FUNCTION_BLOCK FB_FileRingBufferToDB
VAR_INPUT
	udiNovRam_BufferIndex:UDINT;
	udiFile_Index:UDINT;
	dataType:DINT;
END_VAR

IF dataType = E_StructureType.AlarmHistory THEN
	M_AlarmHistory(udiNovRam_BufferIndex:=udiNovRam_BufferIndex,udiFile_Index:=udiFile_Index);
ELSIF dataType = E_StructureType.ProductionHistory THEN
	M_ProductionHistory(udiNovRam_BufferIndex:=udiNovRam_BufferIndex,udiFile_Index:=udiFile_Index);
ELSIF dataType = E_StructureType.ProductionReport THEN
	M_ProductionReport(udiNovRam_BufferIndex:=udiNovRam_BufferIndex,udiFile_Index:=udiFile_Index);
ELSIF dataType = E_StructureType.ProductionSummary THEN
	M_ProductionSummary(udiNovRam_BufferIndex:=udiNovRam_BufferIndex,udiFile_Index:=udiFile_Index);
ELSIF dataType = E_StructureType.SoDuration THEN
	M_SoDuration(udiNovRam_BufferIndex:=udiNovRam_BufferIndex,udiFile_Index:=udiFile_Index);
ELSIF dataType = E_StructureType.StopCount THEN
	M_StopCount(udiNovRam_BufferIndex:=udiNovRam_BufferIndex,udiFile_Index:=udiFile_Index);
ELSIF dataType = E_StructureType.RegularCheckResults THEN
	M_RegularCheckResults(udiNovRam_BufferIndex:=udiNovRam_BufferIndex,udiFile_Index:=udiFile_Index);
END_IF

METHOD M_AlarmHistory : BOOL
VAR_INPUT
	
	//udiFileNo:UDINT;
	udiNovRam_BufferIndex:UDINT;
	udiFile_Index:UDINT;
END_VAR
VAR_INST
	arrDataFromFile:ARRAY[0..GVL.arrArrayLength[E_StructureType.AlarmHistory]-1] OF ST_AlarmInfo_DB_save;
	DataToDB:ST_AlarmInfo_DB_save;
	AnalizeIndex:UDINT;//should be kept by NovRam
	iStep:INT;
	i:UDINT;
	fbFileRingBuffer: FB_FileRingBuffer := ( sNetId     := '',
                                             sPathName  := '',
                                             ePath      := PATH_GENERIC,
                                             nID        := 1,
                                             cbBuffer   := gvl.arrFileRingBufferSize[E_StructureType.AlarmHistory], //5MB(5*10^6Bytes)
                                             bOverwrite := FALSE,
                                             pWriteBuff := 0,
                                             cbWriteLen := 0,
                                             pReadBuff  := 0,
                                             cbReadLen  := 0,
                                             tTimeout   := T#1S );
	bBusy:BOOL;
	bError:BOOL;
	nErrID:UDINT;
	stHeader:ST_FileRBufferHead;
    //loadData  : ARRAY[0..511] OF BYTE :=[512(0)];
    //cbLoad    : UDINT;
	
	fileName: STRING(255);
	eStrIndex:DINT;
	fbAlarmHistory_DB		: FB_AlarmHistory_DB;
END_VAR
//Config
eStrIndex:=E_StructureType.AlarmHistory;

fbFileRingBuffer(sPathName:=fileName
				,bBusy=>bBusy,bError=>bError,nErrID=>nErrID
				,stHeader=>stHeader);
//DB_Test
fbAlarmHistory_DB(udiDBID:=1);

CASE iStep OF
	0://check if file full 
		IF gvl.NovRamData.arrFileRingBuffer_Status[eStrIndex].bFileFull[udiNovRam_BufferIndex][udiFile_Index] = TRUE//file full = should work 
		THEN
			
			fileName:=M_GetFileName(structureType:=eStrIndex
									,udiNovRam_BufferIndex:=udiNovRam_BufferIndex
									,udiFile_Index:=udiFile_Index);
			
			iStep:=100;
		END_IF
	100:// Open file
		
		AnalizeIndex:=0;
		fbFileRingBuffer.A_Open();
		
		iStep:=200;
	200://wait done / read head
		IF NOT fbFileRingBuffer.bBusy AND NOT fbFileRingBuffer.bError THEN
			
			fbFileRingBuffer.A_GetHead(pReadBuff := ADR(arrDataFromFile), cbReadLen := SIZEOF(arrDataFromFile));
			
			iStep:=300;
		END_IF
	300://wait done / take data from array
		IF NOT fbFileRingBuffer.bBusy AND NOT fbFileRingBuffer.bError THEN
			
			DataToDB:=arrDataFromFile[AnalizeIndex];
			
			iStep:=310;
		ELSIF NOT fbFileRingBuffer.bBusy AND fbFileRingBuffer.bError THEN//Empty
			iStep:=600;
		END_IF
	310:// write to DB
	
		//write DataToDB to DB
		DataToDB.lrTime_ms    	:= 987;
		DataToDB.diMsgNumber  	:= 777;
		DataToDB.sTimeString 	:= '2023-11-24 17:17:17';
		DataToDB.wsMsgText    	:= "TEST_MsgText軟體測試";
		DataToDB.sPLC        	:= 'CoreSysTest';
		DataToDB.wsEquipment  	:= "RSA軟體測試";
		DataToDB.sFaam_id    	:= 'TEST_Faam_id';
		
		IF fbAlarmHistory_DB.M_Upload(stAlarmInfo:=DataToDB) THEN
			iStep:=320;
		END_IF
		
	320://wait done
		
		IF NOT fbAlarmHistory_DB.bError THEN//write OK
		
			AnalizeIndex:=AnalizeIndex+1;
			
			iStep:=330;
			
		ELSE//write failed need to write to log
			;
		END_IF
		
	330://Check if all data in array Analized
		IF AnalizeIndex < GVL.arrArrayLength[eStrIndex] THEN//not done
			iStep:=300;//go back
		ELSE//array data done
			iStep:=400;//complete this array
		END_IF
		
	400://wait done / remove Head
	
		fbFileRingBuffer.A_RemoveHead(pReadBuff := ADR(arrDataFromFile), cbReadLen := SIZEOF(arrDataFromFile));
		
		iStep:=500;
		
	500://wait done / check if all data got?
		IF NOT fbFileRingBuffer.bBusy AND NOT fbFileRingBuffer.bError THEN
			IF stHeader.nCount > 0 THEN
				iStep:=100;//Go Back
			ELSE
				iStep:=600;//finish
			END_IF
		END_IF
	600://reset file
	
		fbFileRingBuffer.A_Reset();
		
		iStep:=700;
		
	700://wait done / close file
		IF NOT fbFileRingBuffer.bBusy AND NOT fbFileRingBuffer.bError THEN
			
			fbFileRingBuffer.A_Close();
			
			iStep:=800;
		END_IF
	800://wait done
		IF NOT fbFileRingBuffer.bBusy AND NOT fbFileRingBuffer.bError THEN
			
			GVL.NovRamData.arrFileRingBuffer_Status[eStrIndex].bFileFull[udiNovRam_BufferIndex][udiFile_Index]:=FALSE;
			
			iStep:=0;
			
		END_IF
		
	
END_CASE
END_METHOD

METHOD M_GetFileName : STRING(255)
VAR_INPUT
	structureType:DINT;
	udiNovRam_BufferIndex:UDINT;
	udiFile_Index:UDINT;
END_VAR
VAR
	tempString:STRING(255);
	tempString2:STRING(255);
	tempFileNo:UDINT;
END_VAR
IF structureType=E_StructureType.AlarmHistory THEN
	tempString:=CONCAT(gvl.arrfileFolder[structureType],'AlarmHistory');
ELSIF structureType=E_StructureType.ProductionHistory THEN
	tempString:=CONCAT(gvl.arrfileFolder[structureType],'ProductionHistory');
ELSIF structureType=E_StructureType.ProductionReport THEN
	tempString:=CONCAT(gvl.arrfileFolder[structureType],'ProductionReport');
	ELSIF structureType=E_StructureType.ProductionSummary THEN
	tempString:=CONCAT(gvl.arrfileFolder[structureType],'ProductionSummary');
ELSIF structureType=E_StructureType.SoDuration THEN
	tempString:=CONCAT(gvl.arrfileFolder[structureType],'SoDuration');
ELSIF structureType=E_StructureType.StopCount THEN
	tempString:=CONCAT(gvl.arrfileFolder[structureType],'StopCount');
ELSIF structureType=E_StructureType.RegularCheckResults THEN
	tempString:=CONCAT(gvl.arrfileFolder[structureType],'RegularCheckResults');
END_IF

tempFileNo:=(udiNovRam_BufferIndex) * GVL.FileRingBufferRatio + (udiFile_Index + 1);
tempString2:=CONCAT(tempString,UDINT_TO_STRING(tempFileNo));
M_GetFileName:=CONCAT(tempString2,'.dat');
END_METHOD

{warning 'add method implementation '}
METHOD M_ProductionHistory : BOOL
VAR_INPUT
	
	//udiFileNo:UDINT;
	udiNovRam_BufferIndex:UDINT;
	udiFile_Index:UDINT;
END_VAR
VAR_INST
	arrDataFromFile:ARRAY[0..GVL.arrArrayLength[E_StructureType.ProductionHistory]-1] OF ST_Production_History_DB_Test;
	DataToDB:ST_Production_History_DB_Test;
	AnalizeIndex:UDINT;//should be kept by NovRam
	iStep:INT;
	i:UDINT;
	fbFileRingBuffer: FB_FileRingBuffer := ( sNetId     := '',
                                             sPathName  := '',
                                             ePath      := PATH_GENERIC,
                                             nID        := 1,
                                             cbBuffer   := gvl.arrFileRingBufferSize[E_StructureType.ProductionHistory], //5MB(5*10^6Bytes)
                                             bOverwrite := FALSE,
                                             pWriteBuff := 0,
                                             cbWriteLen := 0,
                                             pReadBuff  := 0,
                                             cbReadLen  := 0,
                                             tTimeout   := T#1S );
	bBusy:BOOL;
	bError:BOOL;
	nErrID:UDINT;
	stHeader:ST_FileRBufferHead;
    //loadData  : ARRAY[0..511] OF BYTE :=[512(0)];
    //cbLoad    : UDINT;
	
	fileName: STRING(255);
	eStrIndex:DINT;
	
	//DB
	fbProductionHistoryInspection_DB		: FB_ProductionHistoryInspection_DB;
	PHI_GroupData_DB : ST_PHI_GroupData_DB;
END_VAR
//Config
eStrIndex:=E_StructureType.ProductionHistory;

fbFileRingBuffer(sPathName:=fileName
				,bBusy=>bBusy,bError=>bError,nErrID=>nErrID
				,stHeader=>stHeader);
				
//DB_Test
fbProductionHistoryInspection_DB(udiDBID:=1);

CASE iStep OF
	0://check if file full 
		IF gvl.NovRamData.arrFileRingBuffer_Status[eStrIndex].bFileFull[udiNovRam_BufferIndex][udiFile_Index] = TRUE//file full = should work 
		THEN
			
			fileName:=M_GetFileName(structureType:=eStrIndex
									,udiNovRam_BufferIndex:=udiNovRam_BufferIndex
									,udiFile_Index:=udiFile_Index);
			
			iStep:=100;
		END_IF
	100:// Open file
		
		AnalizeIndex:=0;
		fbFileRingBuffer.A_Open();
		
		iStep:=200;
	200://wait done / read head
		IF NOT fbFileRingBuffer.bBusy AND NOT fbFileRingBuffer.bError THEN
			
			fbFileRingBuffer.A_GetHead(pReadBuff := ADR(arrDataFromFile), cbReadLen := SIZEOF(arrDataFromFile));
			
			iStep:=300;
		END_IF
	300://wait done / take data from array
		IF NOT fbFileRingBuffer.bBusy AND NOT fbFileRingBuffer.bError THEN
			
			DataToDB:=arrDataFromFile[AnalizeIndex];
			
			iStep:=310;
		ELSIF NOT fbFileRingBuffer.bBusy AND fbFileRingBuffer.bError THEN//Empty
			iStep:=600;
		END_IF
	310:// write to DB
	
		//write DataToDB to DB
		DataToDB.rDuration    	:= 987;
		DataToDB.usiStation_number  	:= 87;
		DataToDB.sStation_name 	:= 'Station Test';
		DataToDB.sFaam_id    	:= 'TEST_Faam_id';
		
		PHI_GroupData_DB.stProductHistory.dtStart_time 			:= TIME_TO_DT(TIME());
		PHI_GroupData_DB.stProductHistory.dtEnd_time 				:= TIME_TO_DT(TIME());
		PHI_GroupData_DB.stProductHistory.rDuration 				:= TIME_TO_REAL(TIME()) / 1000; // ms to s
		PHI_GroupData_DB.stProductHistory.diStation_number 		:= 1;	// index id
		PHI_GroupData_DB.stProductHistory.wsStation_name 			:= "TEST_Station1";		// index name from DB.HC
		PHI_GroupData_DB.stProductHistory.diTrack_number 			:= 1;	//20230106 改為hardcode 1
		PHI_GroupData_DB.stProductHistory.bPart_ok_overal_results := TRUE;
		PHI_GroupData_DB.stProductHistory.sSo_number 				:= 'Fred';				// From ADS  //需要對應DB的So表的So_Number
		PHI_GroupData_DB.stProductHistory.sFaam_id 				:= 'FB000120-E002-0001';		// from DB
		PHI_GroupData_DB.stProductHistory.diSo_id 				:= 3736;			// from ADS  //需要對應DB的So表So_id
		PHI_GroupData_DB.stProductHistory.diWpc_number			:= 2; // ShuttleID
		
		IF fbProductionHistoryInspection_DB.M_Upload(stPHI:=PHI_GroupData_DB) THEN
			iStep:=320;
		END_IF
		
	320://wait done
		
		IF NOT fbProductionHistoryInspection_DB.bError THEN//write OK
		
			AnalizeIndex:=AnalizeIndex+1;
			
			iStep:=330;
			
		ELSE//write failed need to write to log
			;
		END_IF
		
	330://Check if all data in array Analized
		IF AnalizeIndex < GVL.arrArrayLength[eStrIndex] THEN//not done
			iStep:=300;//go back
		ELSE//array data done
			iStep:=400;//complete this array
		END_IF
		
	400://wait done / remove Head
	
		fbFileRingBuffer.A_RemoveHead(pReadBuff := ADR(arrDataFromFile), cbReadLen := SIZEOF(arrDataFromFile));
		
		iStep:=500;
		
	500://wait done / check if all data got?
		IF NOT fbFileRingBuffer.bBusy AND NOT fbFileRingBuffer.bError THEN
			IF stHeader.nCount > 0 THEN
				iStep:=100;//Go Back
			ELSE
				iStep:=600;//finish
			END_IF
		END_IF
	600://reset file
	
		fbFileRingBuffer.A_Reset();
		
		iStep:=700;
		
	700://wait done / close file
		IF NOT fbFileRingBuffer.bBusy AND NOT fbFileRingBuffer.bError THEN
			
			fbFileRingBuffer.A_Close();
			
			iStep:=800;
		END_IF
	800://wait done
		IF NOT fbFileRingBuffer.bBusy AND NOT fbFileRingBuffer.bError THEN
			
			GVL.NovRamData.arrFileRingBuffer_Status[eStrIndex].bFileFull[udiNovRam_BufferIndex][udiFile_Index]:=FALSE;
			
			iStep:=0;
			
		END_IF
		
	
END_CASE
END_METHOD

METHOD M_ProductionReport : BOOL
VAR_INPUT
	
	//udiFileNo:UDINT;
	udiNovRam_BufferIndex:UDINT;
	udiFile_Index:UDINT;
END_VAR
VAR_INST
	arrDataFromFile:ARRAY[0..GVL.arrArrayLength[E_StructureType.ProductionReport]-1] OF ST_OEE_ProductionReport;
	DataToDB:ST_OEE_ProductionReport;
	AnalizeIndex:UDINT;//should be kept by NovRam
	iStep:INT;
	i:UDINT;
	fbFileRingBuffer: FB_FileRingBuffer := ( sNetId     := '',
                                             sPathName  := '',
                                             ePath      := PATH_GENERIC,
                                             nID        := 1,
                                             cbBuffer   := gvl.arrFileRingBufferSize[E_StructureType.ProductionReport], //5MB(5*10^6Bytes)
                                             bOverwrite := FALSE,
                                             pWriteBuff := 0,
                                             cbWriteLen := 0,
                                             pReadBuff  := 0,
                                             cbReadLen  := 0,
                                             tTimeout   := T#1S );
	bBusy:BOOL;
	bError:BOOL;
	nErrID:UDINT;
	stHeader:ST_FileRBufferHead;
    //loadData  : ARRAY[0..511] OF BYTE :=[512(0)];
    //cbLoad    : UDINT;
	
	fileName: STRING(255);
	eStrIndex:DINT;
	fbOEE_ProductionReport_DB:FB_OEE_ProductionReport_DB;
END_VAR
//Config
eStrIndex:=E_StructureType.ProductionReport;

fbFileRingBuffer(sPathName:=fileName
				,bBusy=>bBusy,bError=>bError,nErrID=>nErrID
				,stHeader=>stHeader);
				
CASE iStep OF
	0://check if file full 
		IF gvl.NovRamData.arrFileRingBuffer_Status[eStrIndex].bFileFull[udiNovRam_BufferIndex][udiFile_Index] = TRUE//file full = should work 
		THEN
			
			fileName:=M_GetFileName(structureType:=eStrIndex
									,udiNovRam_BufferIndex:=udiNovRam_BufferIndex
									,udiFile_Index:=udiFile_Index);
			
			iStep:=100;
		END_IF
	100:// Open file
		
		AnalizeIndex:=0;
		fbFileRingBuffer.A_Open();
		
		iStep:=200;
	200://wait done / read head
		IF NOT fbFileRingBuffer.bBusy AND NOT fbFileRingBuffer.bError THEN
			
			fbFileRingBuffer.A_GetHead(pReadBuff := ADR(arrDataFromFile), cbReadLen := SIZEOF(arrDataFromFile));
			
			iStep:=300;
		END_IF
	300://wait done / take data from array
		IF NOT fbFileRingBuffer.bBusy AND NOT fbFileRingBuffer.bError THEN
			
			DataToDB:=arrDataFromFile[AnalizeIndex];
			
			iStep:=310;
		ELSIF NOT fbFileRingBuffer.bBusy AND fbFileRingBuffer.bError THEN//Empty
			iStep:=600;
		END_IF
	310:// write to DB
	
		//write DataToDB to DB
		DataToDB.diOk_part_count:=123;
		DataToDB.sSo_number                    	:= 'Fred';
		DataToDB.sFaam_id                      	:= 'FB000120-E002-0001';
		DataToDB.diSo_id                        := 3736;
		
		IF fbOEE_ProductionReport_DB.M_Upload(stOeeProductionReport:=DataToDB) THEN
			iStep:=320;
		END_IF
		
	320://wait done
		
			IF NOT fbOEE_ProductionReport_DB.bError THEN//write OK
			
				AnalizeIndex:=AnalizeIndex+1;
				
				iStep:=330;
				
			ELSE//write failed need to write to log
				;
			END_IF
		
		
	330://Check if all data in array Analized
		IF AnalizeIndex < GVL.arrArrayLength[eStrIndex] THEN//not done
			iStep:=300;//go back
		ELSE//array data done
			iStep:=400;//complete this array
		END_IF
		
	400://wait done / remove Head
	
		fbFileRingBuffer.A_RemoveHead(pReadBuff := ADR(arrDataFromFile), cbReadLen := SIZEOF(arrDataFromFile));
		
		iStep:=500;
		
	500://wait done / check if all data got?
		IF NOT fbFileRingBuffer.bBusy AND NOT fbFileRingBuffer.bError THEN
			IF stHeader.nCount > 0 THEN
				iStep:=100;//Go Back
			ELSE
				iStep:=600;//finish
			END_IF
		END_IF
	600://reset file
	
		fbFileRingBuffer.A_Reset();
		
		iStep:=700;
		
	700://wait done / close file
		IF NOT fbFileRingBuffer.bBusy AND NOT fbFileRingBuffer.bError THEN
			
			fbFileRingBuffer.A_Close();
			
			iStep:=800;
		END_IF
	800://wait done
		IF NOT fbFileRingBuffer.bBusy AND NOT fbFileRingBuffer.bError THEN
			
			GVL.NovRamData.arrFileRingBuffer_Status[eStrIndex].bFileFull[udiNovRam_BufferIndex][udiFile_Index]:=FALSE;
			
			iStep:=0;
			
		END_IF
		
	
END_CASE
END_METHOD

METHOD M_ProductionSummary : BOOL
VAR_INPUT
	
	//udiFileNo:UDINT;
	udiNovRam_BufferIndex:UDINT;
	udiFile_Index:UDINT;
END_VAR
VAR_INST
	arrDataFromFile:ARRAY[0..GVL.arrArrayLength[E_StructureType.ProductionSummary]-1] OF ST_OEE_ProductionSummary;
	DataToDB:ST_OEE_ProductionSummary;
	AnalizeIndex:UDINT;//should be kept by NovRam
	iStep:INT;
	i:UDINT;
	fbFileRingBuffer: FB_FileRingBuffer := ( sNetId     := '',
                                             sPathName  := '',
                                             ePath      := PATH_GENERIC,
                                             nID        := 1,
                                             cbBuffer   := gvl.arrFileRingBufferSize[E_StructureType.ProductionSummary], //5MB(5*10^6Bytes)
                                             bOverwrite := FALSE,
                                             pWriteBuff := 0,
                                             cbWriteLen := 0,
                                             pReadBuff  := 0,
                                             cbReadLen  := 0,
                                             tTimeout   := T#1S );
	bBusy:BOOL;
	bError:BOOL;
	nErrID:UDINT;
	stHeader:ST_FileRBufferHead;
    //loadData  : ARRAY[0..511] OF BYTE :=[512(0)];
    //cbLoad    : UDINT;
	
	fileName: STRING(255);
	eStrIndex:DINT;
	fbOEE_ProductionSummary_DB:FB_OEE_ProductionSummary_DB;
END_VAR
//Config
eStrIndex:=E_StructureType.ProductionSummary;

fbFileRingBuffer(sPathName:=fileName
				,bBusy=>bBusy,bError=>bError,nErrID=>nErrID
				,stHeader=>stHeader);
				
CASE iStep OF
	0://check if file full 
		IF gvl.NovRamData.arrFileRingBuffer_Status[eStrIndex].bFileFull[udiNovRam_BufferIndex][udiFile_Index] = TRUE//file full = should work 
		THEN
			
			fileName:=M_GetFileName(structureType:=eStrIndex
									,udiNovRam_BufferIndex:=udiNovRam_BufferIndex
									,udiFile_Index:=udiFile_Index);
			
			iStep:=100;
		END_IF
	100:// Open file
		
		AnalizeIndex:=0;
		fbFileRingBuffer.A_Open();
		
		iStep:=200;
	200://wait done / read head
		IF NOT fbFileRingBuffer.bBusy AND NOT fbFileRingBuffer.bError THEN
			
			fbFileRingBuffer.A_GetHead(pReadBuff := ADR(arrDataFromFile), cbReadLen := SIZEOF(arrDataFromFile));
			
			iStep:=300;
		END_IF
	300://wait done / take data from array
		IF NOT fbFileRingBuffer.bBusy AND NOT fbFileRingBuffer.bError THEN
			
			DataToDB:=arrDataFromFile[AnalizeIndex];
			
			iStep:=310;
		ELSIF NOT fbFileRingBuffer.bBusy AND fbFileRingBuffer.bError THEN//Empty
			iStep:=600;
		END_IF
	310:// write to DB
	
		//write DataToDB to DB
		DataToDB.diSo_id:=123;
		DataToDB.diSummary_value:=456;
		DataToDB.sSo_number                    	:= 'Fred';
		DataToDB.sFaam_id                      	:= 'FB000120-E002-0001';
		DataToDB.diSo_id                        := 3736;
		
		IF fbOEE_ProductionSummary_DB.M_Upload(stOEEProductionSummary:=DataToDB) THEN
			iStep:=320;
		END_IF
		
		
	320://wait done
		
			IF NOT fbOEE_ProductionSummary_DB.bError THEN//write OK
			
				AnalizeIndex:=AnalizeIndex+1;
				
				iStep:=330;
				
			ELSE//write failed need to write to log
				;
			END_IF
		
		
	330://Check if all data in array Analized
		IF AnalizeIndex < GVL.arrArrayLength[eStrIndex] THEN//not done
			iStep:=300;//go back
		ELSE//array data done
			iStep:=400;//complete this array
		END_IF
		
	400://wait done / remove Head
	
		fbFileRingBuffer.A_RemoveHead(pReadBuff := ADR(arrDataFromFile), cbReadLen := SIZEOF(arrDataFromFile));
		
		iStep:=500;
		
	500://wait done / check if all data got?
		IF NOT fbFileRingBuffer.bBusy AND NOT fbFileRingBuffer.bError THEN
			IF stHeader.nCount > 0 THEN
				iStep:=100;//Go Back
			ELSE
				iStep:=600;//finish
			END_IF
		END_IF
	600://reset file
	
		fbFileRingBuffer.A_Reset();
		
		iStep:=700;
		
	700://wait done / close file
		IF NOT fbFileRingBuffer.bBusy AND NOT fbFileRingBuffer.bError THEN
			
			fbFileRingBuffer.A_Close();
			
			iStep:=800;
		END_IF
	800://wait done
		IF NOT fbFileRingBuffer.bBusy AND NOT fbFileRingBuffer.bError THEN
			
			GVL.NovRamData.arrFileRingBuffer_Status[eStrIndex].bFileFull[udiNovRam_BufferIndex][udiFile_Index]:=FALSE;
			
			iStep:=0;
			
		END_IF
		
	
END_CASE
END_METHOD

METHOD M_RegularCheckResults : BOOL
VAR_INPUT
	
	//udiFileNo:UDINT;
	udiNovRam_BufferIndex:UDINT;
	udiFile_Index:UDINT;
END_VAR
VAR_INST
	arrDataFromFile:ARRAY[0..GVL.arrArrayLength[E_StructureType.RegularCheckResults]-1] OF ST_RegularCheck_Results_DB;
	DataToDB:ST_RegularCheck_Results;//TEST
	AnalizeIndex:UDINT;//should be kept by NovRam
	iStep:INT;
	i:UDINT;
	fbFileRingBuffer: FB_FileRingBuffer := ( sNetId     := '',
                                             sPathName  := '',
                                             ePath      := PATH_GENERIC,
                                             nID        := 1,
                                             cbBuffer   := gvl.arrFileRingBufferSize[E_StructureType.RegularCheckResults], //5MB(5*10^6Bytes)
                                             bOverwrite := FALSE,
                                             pWriteBuff := 0,
                                             cbWriteLen := 0,
                                             pReadBuff  := 0,
                                             cbReadLen  := 0,
                                             tTimeout   := T#1S );
	bBusy:BOOL;
	bError:BOOL;
	nErrID:UDINT;
	stHeader:ST_FileRBufferHead;
    //loadData  : ARRAY[0..511] OF BYTE :=[512(0)];
    //cbLoad    : UDINT;
	
	fileName: STRING(255);
	eStrIndex:DINT;
	fbRegular_Check_Results_DB:FB_Regular_Check_Results_DB;
END_VAR
//Config
eStrIndex:=E_StructureType.RegularCheckResults;

fbFileRingBuffer(sPathName:=fileName
				,bBusy=>bBusy,bError=>bError,nErrID=>nErrID
				,stHeader=>stHeader);
				
CASE iStep OF
	0://check if file full 
		IF gvl.NovRamData.arrFileRingBuffer_Status[eStrIndex].bFileFull[udiNovRam_BufferIndex][udiFile_Index] = TRUE//file full = should work 
		THEN
			
			fileName:=M_GetFileName(structureType:=eStrIndex
									,udiNovRam_BufferIndex:=udiNovRam_BufferIndex
									,udiFile_Index:=udiFile_Index);
			
			iStep:=100;
		END_IF
	100:// Open file
		
		AnalizeIndex:=0;
		fbFileRingBuffer.A_Open();
		
		iStep:=200;
	200://wait done / read head
		IF NOT fbFileRingBuffer.bBusy AND NOT fbFileRingBuffer.bError THEN
			
			fbFileRingBuffer.A_GetHead(pReadBuff := ADR(arrDataFromFile), cbReadLen := SIZEOF(arrDataFromFile));
			
			iStep:=300;
		END_IF
	300://wait done / take data from array
		IF NOT fbFileRingBuffer.bBusy AND NOT fbFileRingBuffer.bError THEN
			
			//DataToDB:=arrDataFromFile[AnalizeIndex];
			M_ST_RegularCheckResults_Convert(input:=arrDataFromFile[AnalizeIndex]
											,output=>DataToDB);
			iStep:=310;
		ELSIF NOT fbFileRingBuffer.bBusy AND fbFileRingBuffer.bError THEN//Empty
			iStep:=600;
		END_IF
	310:// write to DB
		
		//write DataToDB to DB
		DataToDB.eSensor:=E_RegularCheckSensorResult.Fail;
		DataToDB.eSensor2:=E_RegularCheckSensorResult.Fail;
		DataToDB.sSo_number                    	:= 'Fred';
		DataToDB.sFaam_id                      	:= 'FB000120-E002-0001';
		DataToDB.diSo_id                        := 3736;
		
		IF fbRegular_Check_Results_DB.M_Upload(stRcResults:=DataToDB) THEN
			iStep:=320;
		END_IF
		
	320://wait done
		
		IF NOT fbRegular_Check_Results_DB.bError THEN//write OK
		
			AnalizeIndex:=AnalizeIndex+1;
			
			iStep:=330;
			
		ELSE//write failed need to write to log
			;
		END_IF
		
	330://Check if all data in array Analized
		IF AnalizeIndex < GVL.arrArrayLength[eStrIndex] THEN//not done
			iStep:=300;//go back
		ELSE//array data done
			iStep:=400;//complete this array
		END_IF
		
	400://wait done / remove Head
	
		fbFileRingBuffer.A_RemoveHead(pReadBuff := ADR(arrDataFromFile), cbReadLen := SIZEOF(arrDataFromFile));
		
		iStep:=500;
		
	500://wait done / check if all data got?
		IF NOT fbFileRingBuffer.bBusy AND NOT fbFileRingBuffer.bError THEN
			IF stHeader.nCount > 0 THEN
				iStep:=100;//Go Back
			ELSE
				iStep:=600;//finish
			END_IF
		END_IF
	600://reset file
	
		fbFileRingBuffer.A_Reset();
		
		iStep:=700;
		
	700://wait done / close file
		IF NOT fbFileRingBuffer.bBusy AND NOT fbFileRingBuffer.bError THEN
			
			fbFileRingBuffer.A_Close();
			
			iStep:=800;
		END_IF
	800://wait done
		IF NOT fbFileRingBuffer.bBusy AND NOT fbFileRingBuffer.bError THEN
			
			GVL.NovRamData.arrFileRingBuffer_Status[eStrIndex].bFileFull[udiNovRam_BufferIndex][udiFile_Index]:=FALSE;
			
			iStep:=0;
			
		END_IF
		
	
END_CASE
END_METHOD

METHOD M_SoDuration : BOOL
VAR_INPUT
	
	//udiFileNo:UDINT;
	udiNovRam_BufferIndex:UDINT;
	udiFile_Index:UDINT;
END_VAR
VAR_INST
	arrDataFromFile:ARRAY[0..GVL.arrArrayLength[E_StructureType.SoDuration]-1] OF ST_SoDuration;
	DataToDB:ST_SoDuration;
	AnalizeIndex:UDINT;//should be kept by NovRam
	iStep:INT;
	i:UDINT;
	fbFileRingBuffer: FB_FileRingBuffer := ( sNetId     := '',
                                             sPathName  := '',
                                             ePath      := PATH_GENERIC,
                                             nID        := 1,
                                             cbBuffer   := gvl.arrFileRingBufferSize[E_StructureType.ProductionSummary], //5MB(5*10^6Bytes)
                                             bOverwrite := FALSE,
                                             pWriteBuff := 0,
                                             cbWriteLen := 0,
                                             pReadBuff  := 0,
                                             cbReadLen  := 0,
                                             tTimeout   := T#1S );
	bBusy:BOOL;
	bError:BOOL;
	nErrID:UDINT;
	stHeader:ST_FileRBufferHead;
    //loadData  : ARRAY[0..511] OF BYTE :=[512(0)];
    //cbLoad    : UDINT;
	
	fileName: STRING(255);
	eStrIndex:DINT;
	fbSoDuration_DB:FB_SoDuration_DB;
	
END_VAR
//Config
eStrIndex:=E_StructureType.SoDuration;

fbFileRingBuffer(sPathName:=fileName
				,bBusy=>bBusy,bError=>bError,nErrID=>nErrID
				,stHeader=>stHeader);
				
CASE iStep OF
	0://check if file full 
		IF gvl.NovRamData.arrFileRingBuffer_Status[eStrIndex].bFileFull[udiNovRam_BufferIndex][udiFile_Index] = TRUE//file full = should work 
		THEN
			
			fileName:=M_GetFileName(structureType:=eStrIndex
									,udiNovRam_BufferIndex:=udiNovRam_BufferIndex
									,udiFile_Index:=udiFile_Index);
			
			iStep:=100;
		END_IF
	100:// Open file
		
		AnalizeIndex:=0;
		fbFileRingBuffer.A_Open();
		
		iStep:=200;
	200://wait done / read head
		IF NOT fbFileRingBuffer.bBusy AND NOT fbFileRingBuffer.bError THEN
			
			fbFileRingBuffer.A_GetHead(pReadBuff := ADR(arrDataFromFile), cbReadLen := SIZEOF(arrDataFromFile));
			
			iStep:=300;
		END_IF
	300://wait done / take data from array
		IF NOT fbFileRingBuffer.bBusy AND NOT fbFileRingBuffer.bError THEN
			
			DataToDB:=arrDataFromFile[AnalizeIndex];
			
			iStep:=310;
		ELSIF NOT fbFileRingBuffer.bBusy AND fbFileRingBuffer.bError THEN//Empty
			iStep:=600;
		END_IF
	310:// write to DB
	
		//write DataToDB to DB
		DataToDB.sSo_number                    	:= 'Fred';
		DataToDB.sFaam_id                      	:= 'FB000120-E002-0001';
		DataToDB.diSo_id                        := 3736;
		
		IF fbSoDuration_DB.M_Upload(stSoDuration:=DataToDB) THEN
			iStep:=320;
		END_IF
		
	320://wait done
		
		IF NOT fbSoDuration_DB.bError THEN//write OK
		
			AnalizeIndex:=AnalizeIndex+1;
			
			iStep:=330;
			
		ELSE//write failed need to write to log
			;
		END_IF
		
	330://Check if all data in array Analized
		IF AnalizeIndex < GVL.arrArrayLength[eStrIndex] THEN//not done
			iStep:=300;//go back
		ELSE//array data done
			iStep:=400;//complete this array
		END_IF
		
	400://wait done / remove Head
	
		fbFileRingBuffer.A_RemoveHead(pReadBuff := ADR(arrDataFromFile), cbReadLen := SIZEOF(arrDataFromFile));
		
		iStep:=500;
		
	500://wait done / check if all data got?
		IF NOT fbFileRingBuffer.bBusy AND NOT fbFileRingBuffer.bError THEN
			IF stHeader.nCount > 0 THEN
				iStep:=100;//Go Back
			ELSE
				iStep:=600;//finish
			END_IF
		END_IF
	600://reset file
	
		fbFileRingBuffer.A_Reset();
		
		iStep:=700;
		
	700://wait done / close file
		IF NOT fbFileRingBuffer.bBusy AND NOT fbFileRingBuffer.bError THEN
			
			fbFileRingBuffer.A_Close();
			
			iStep:=800;
		END_IF
	800://wait done
		IF NOT fbFileRingBuffer.bBusy AND NOT fbFileRingBuffer.bError THEN
			
			GVL.NovRamData.arrFileRingBuffer_Status[eStrIndex].bFileFull[udiNovRam_BufferIndex][udiFile_Index]:=FALSE;
			
			iStep:=0;
			
		END_IF
		
	
END_CASE
END_METHOD

METHOD M_ST_AlarmHistory_Convert : BOOL
VAR_INPUT
END_VAR
END_METHOD

METHOD M_ST_ProductionHistory_Convert : BOOL
VAR_INPUT
END_VAR
END_METHOD

METHOD M_ST_ProductionReport_Convert : BOOL
VAR_INPUT
END_VAR
END_METHOD

METHOD M_ST_ProductionSummary_Convert : BOOL
VAR_INPUT
END_VAR
END_METHOD

METHOD M_ST_RegularCheckResults_Convert : BOOL
VAR_INPUT
	input:ST_RegularCheck_Results_DB;
END_VAR
VAR_OUTPUT
	output:ST_RegularCheck_Results;
END_VAR
END_METHOD

METHOD M_ST_SoDuration_Convert : BOOL
VAR_INPUT
END_VAR
END_METHOD

METHOD M_ST_StopCount_Convert : BOOL
VAR_INPUT
END_VAR
END_METHOD

METHOD M_StopCount : BOOL
VAR_INPUT
	
	//udiFileNo:UDINT;
	udiNovRam_BufferIndex:UDINT;
	udiFile_Index:UDINT;
END_VAR
VAR_INST
	arrDataFromFile:ARRAY[0..GVL.arrArrayLength[E_StructureType.StopCount]-1] OF ST_StopCount;
	DataToDB:ST_StopCount;
	AnalizeIndex:UDINT;//should be kept by NovRam
	iStep:INT;
	i:UDINT;
	fbFileRingBuffer: FB_FileRingBuffer := ( sNetId     := '',
                                             sPathName  := '',
                                             ePath      := PATH_GENERIC,
                                             nID        := 1,
                                             cbBuffer   := gvl.arrFileRingBufferSize[E_StructureType.StopCount], //5MB(5*10^6Bytes)
                                             bOverwrite := FALSE,
                                             pWriteBuff := 0,
                                             cbWriteLen := 0,
                                             pReadBuff  := 0,
                                             cbReadLen  := 0,
                                             tTimeout   := T#1S );
	bBusy:BOOL;
	bError:BOOL;
	nErrID:UDINT;
	stHeader:ST_FileRBufferHead;
    //loadData  : ARRAY[0..511] OF BYTE :=[512(0)];
    //cbLoad    : UDINT;
	
	fileName: STRING(255);
	eStrIndex:DINT;
	fbStopCount_DB:FB_StopCount_DB;
END_VAR
//Config
eStrIndex:=E_StructureType.StopCount;

fbFileRingBuffer(sPathName:=fileName
				,bBusy=>bBusy,bError=>bError,nErrID=>nErrID
				,stHeader=>stHeader);
				
CASE iStep OF
	0://check if file full 
		IF gvl.NovRamData.arrFileRingBuffer_Status[eStrIndex].bFileFull[udiNovRam_BufferIndex][udiFile_Index] = TRUE//file full = should work 
		THEN
			
			fileName:=M_GetFileName(structureType:=eStrIndex
									,udiNovRam_BufferIndex:=udiNovRam_BufferIndex
									,udiFile_Index:=udiFile_Index);
			
			iStep:=100;
		END_IF
	100:// Open file
		
		AnalizeIndex:=0;
		fbFileRingBuffer.A_Open();
		
		iStep:=200;
	200://wait done / read head
		IF NOT fbFileRingBuffer.bBusy AND NOT fbFileRingBuffer.bError THEN
			
			fbFileRingBuffer.A_GetHead(pReadBuff := ADR(arrDataFromFile), cbReadLen := SIZEOF(arrDataFromFile));
			
			iStep:=300;
		END_IF
	300://wait done / take data from array
		IF NOT fbFileRingBuffer.bBusy AND NOT fbFileRingBuffer.bError THEN
			
			DataToDB:=arrDataFromFile[AnalizeIndex];
			
			iStep:=310;
		ELSIF NOT fbFileRingBuffer.bBusy AND fbFileRingBuffer.bError THEN//Empty
			iStep:=600;
		END_IF
	310:// write to DB
		
		//write DataToDB to DB
		DataToDB.sSo_number                    	:= 'Fred';
		DataToDB.sFaam_id                      	:= 'FB000120-E002-0001';
		DataToDB.diSo_id                        := 3736;
		
		IF fbStopCount_DB.M_Upload(stStopCount:=DataToDB) THEN
			iStep:=320;
		END_IF
		
	320://wait done
		
		IF NOT fbStopCount_DB.bError THEN//write OK
		
			AnalizeIndex:=AnalizeIndex+1;
			
			iStep:=330;
			
		ELSE//write failed need to write to log
			;
		END_IF
		
	330://Check if all data in array Analized
		IF AnalizeIndex < GVL.arrArrayLength[eStrIndex] THEN//not done
			iStep:=300;//go back
		ELSE//array data done
			iStep:=400;//complete this array
		END_IF
		
	400://wait done / remove Head
	
		fbFileRingBuffer.A_RemoveHead(pReadBuff := ADR(arrDataFromFile), cbReadLen := SIZEOF(arrDataFromFile));
		
		iStep:=500;
		
	500://wait done / check if all data got?
		IF NOT fbFileRingBuffer.bBusy AND NOT fbFileRingBuffer.bError THEN
			IF stHeader.nCount > 0 THEN
				iStep:=100;//Go Back
			ELSE
				iStep:=600;//finish
			END_IF
		END_IF
	600://reset file
	
		fbFileRingBuffer.A_Reset();
		
		iStep:=700;
		
	700://wait done / close file
		IF NOT fbFileRingBuffer.bBusy AND NOT fbFileRingBuffer.bError THEN
			
			fbFileRingBuffer.A_Close();
			
			iStep:=800;
		END_IF
	800://wait done
		IF NOT fbFileRingBuffer.bBusy AND NOT fbFileRingBuffer.bError THEN
			
			GVL.NovRamData.arrFileRingBuffer_Status[eStrIndex].bFileFull[udiNovRam_BufferIndex][udiFile_Index]:=FALSE;
			
			iStep:=0;
			
		END_IF
		
	
END_CASE
END_METHOD

END_FUNCTION_BLOCK

(* stored: Version 1.1.0.1, ProductVersion 3.1.4024.11
   POU FB_FileRingBufferToDB: Id {5407df28-5241-4688-9419-685e8c9548d2}, SpecialFunc None
   Folder Sub: Id {2534213c-7e5e-4abf-9411-860d44a5b2d2}
   Method M_AlarmHistory: Id {ff77384c-01f1-48bd-a1b3-7abc9b26720b}
   Method M_GetFileName: Id {4b3fabe7-1e25-46e4-9798-bee9befa9ab6}
   Method M_ProductionHistory: Id {8fa7d530-7099-445c-bf55-d19dcfd86a46}
   Method M_ProductionReport: Id {50ec54d4-867e-4233-ac7e-27f8467d1362}
   Method M_ProductionSummary: Id {cc4bac99-b6fb-4a33-86fa-fb65566bf866}
   Method M_RegularCheckResults: Id {c1a33c14-6851-44f5-b745-cb1a1bc9c7c4}
   Method M_SoDuration: Id {56393071-2555-404b-aac1-71b9d39a0087}
   Method M_ST_AlarmHistory_Convert: Id {90234377-5e57-4a9c-9b48-a547d1d556f7}
   Method M_ST_ProductionHistory_Convert: Id {56b298ca-fed2-4f78-8add-9ff8f9eca520}
   Method M_ST_ProductionReport_Convert: Id {6448b315-2048-49f6-b778-7e67bf20eea8}
   Method M_ST_ProductionSummary_Convert: Id {8cecd652-1a50-4b26-88c4-1513f9101c97}
   Method M_ST_RegularCheckResults_Convert: Id {3d691fe0-8452-4cec-baed-830d96336e29}
   Method M_ST_SoDuration_Convert: Id {8efca6c8-584d-46e0-9bd4-7ed0f3c98d6e}
   Method M_ST_StopCount_Convert: Id {483d237d-5099-4da3-9f28-7308f5bcf526}
   Method M_StopCount: Id {ce4c351f-2ecd-476b-900a-3eebce8b4087} *)
